PROGRAM prgLab02
VAR
	contadorUp:CTU;
	contUp: BOOL;
	resetCount: BOOL;
	countFinished: BOOL;
	counterV: WORD;
	
	trig:R_TRIG;
	bTrigCnt:BOOL;
	contagemAtual:UDINT;
	
	passoContagem: UDINT:=1;
	fimContagem: BOOL;

	contagemProgramada: UDINT:=5;
	
	di1 AT %I*:BOOL;
	do1 AT %Q*:BOOL;
	do2 AT %Q*:BOOL;
	entradaAnalogica AT %I*:INT;
END_VAR
VAR CONSTANT
	var5Volts :INT:=16383;	//32767/2
END_VAR

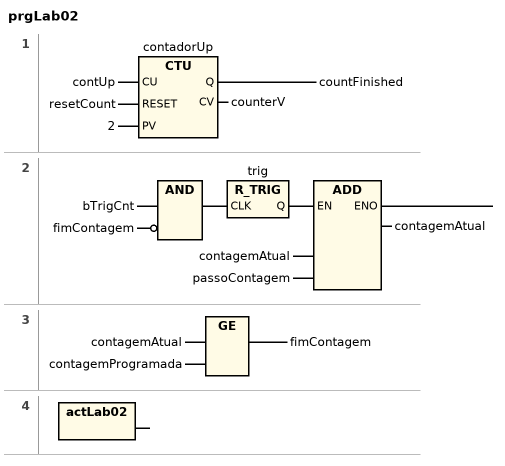
// NETWORK 1
contadorUp(CU := contUp, RESET := resetCount, PV := 2, CV => counterV); // CTU
countFinished := contadorUp.Q;

// NETWORK 2
trig(CLK := bTrigCnt AND NOT fimContagem); // R_TRIG
IF trig.Q THEN contagemAtual := contagemAtual + passoContagem; END_IF

// NETWORK 3
fimContagem := contagemAtual >= contagemProgramada;

// NETWORK 4
actLab02();

ACTION actLab02:
IF di1 THEN
	do1 := entradaAnalogica>= var5Volts;
	do2:= NOT do1;
ELSIF NOT di1 THEN
	do2 := entradaAnalogica>= var5Volts;
	do1:= NOT do2;		
END_IF
END_ACTION

END_PROGRAM

(* stored: Version 1.1.0.1, ProductVersion 3.1.4024.12
   POU prgLab02: Id {b8fb7635-0598-4341-ab31-ace300adc7d5}, SpecialFunc None
   Action actLab02: Id {00615974-0ce5-4184-8a33-de8597686392} *)
